TEXTLIST TextList_Evap
  0 = '' | FR: 'Creuset' | EN: 'Crucible'
  1 = '' | FR: 'Balayage' | EN: 'Sweeping'
  2 = '' | FR: 'Courant' | EN: 'Current'
  3 = '' | FR: 'Haute Tension' | EN: 'High Voltage'
  4 = '' | FR: 'Consigne' | EN: 'Setpoint'
  5 = 'Etat' | FR: 'Etat' | EN: 'State'
   = ''
END_TEXTLIST

(* stored: Version 1.1.0.1, ProductVersion 3.1.4024.10
   TextList TextList_Evap: Id {32d2e278-abd6-4402-9f0a-cd64de10028c} *)
